FUNCTION_BLOCK EL2084
VAR
	{attribute addProperty Name "WcState"}
	_wcState : WcStateInputToggle;
	{attribute addProperty Name "Info data"}
	_infoData : InfoDataAds;
	_io : EL2xx4_Data;
END_VAR

PROPERTY IO : REFERENCE TO EL2xx4_Data
GET
IO REF= _io;
END_GET
END_PROPERTY

PROPERTY WcState : REFERENCE TO WcStateBase
GET
WcState REF= _wcState;
END_GET
END_PROPERTY

END_FUNCTION_BLOCK

(* stored: Version 1.1.0.1, ProductVersion 3.1.4024.9
   POU EL2084: Id {978e746a-b722-0fae-2aae-eeb19061a419}, SpecialFunc None
   Property IO: Id {644c27ce-ef9d-00eb-3237-312495313080}
   Get Get: Id {57b3f45e-dc68-07d6-2f19-1c5aa9f3058e}
   Property WcState: Id {304da218-29ee-0e4c-2d04-3871d45a1f60}
   Get Get: Id {78497d8c-2860-0bf2-3dad-184b268cc580} *)
